
// ===== library types =====

TYPE "ecco"
   STRUCT
      test : Bool;
      "type" : Byte;
      copy : String;
   END_STRUCT;
END_TYPE

FUNCTION_BLOCK "FB-Tipo"   // FB1, LAD
{ S7_Optimized_Access := 'TRUE' }
VERSION : 0.1
BEGIN

REGION Network 1
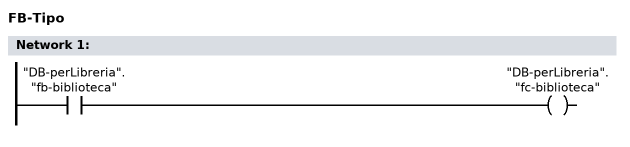
   RUNG wire#powerrail
      Contact( "DB-perLibreria"."fb-biblioteca" )
      Coil( "DB-perLibreria"."fc-biblioteca" )
   END_RUNG
   // the same network as SCL:
   "DB-perLibreria"."fc-biblioteca" := "DB-perLibreria"."fb-biblioteca";
END_REGION
END_FUNCTION_BLOCK

FUNCTION "FC-Tipo" : Void   // FC1, LAD
{ S7_Optimized_Access := 'TRUE' }
VERSION : 0.1
BEGIN

REGION Network 1
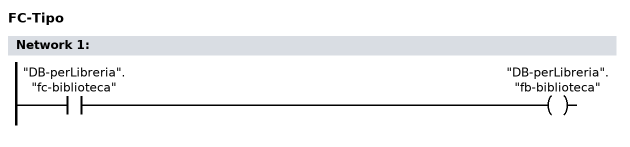
   RUNG wire#powerrail
      Contact( "DB-perLibreria"."fc-biblioteca" )
      Coil( "DB-perLibreria"."fb-biblioteca" )
   END_RUNG
   // the same network as SCL:
   "DB-perLibreria"."fb-biblioteca" := "DB-perLibreria"."fc-biblioteca";
END_REGION
END_FUNCTION

// ===== library: MasterCopy "DB-inLibreria" =====

DATA_BLOCK "DB-perLibreria"   // DB2
{ S7_Optimized_Access := 'TRUE' }
VERSION : 0.1
   VAR
      "fb-biblioteca" : Bool;
      "fc-biblioteca" : Bool;
      prova : "ecco";
   END_VAR
BEGIN
END_DATA_BLOCK

// ===== library: MasterCopy "FB-inLibreria" =====

FUNCTION_BLOCK "FB-inLibreria"   // FB1, LAD
{ S7_Optimized_Access := 'TRUE' }
VERSION : 0.1
BEGIN

REGION Network 1
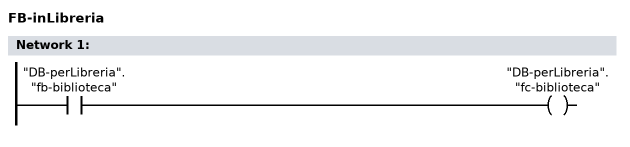
   RUNG wire#powerrail
      Contact( "DB-perLibreria"."fb-biblioteca" )
      Coil( "DB-perLibreria"."fc-biblioteca" )
   END_RUNG
   // the same network as SCL:
   "DB-perLibreria"."fc-biblioteca" := "DB-perLibreria"."fb-biblioteca";
END_REGION
END_FUNCTION_BLOCK

// ===== library: MasterCopy "FC-inLibreria" =====

FUNCTION "FC-inLibreria" : Void   // FC1, LAD
{ S7_Optimized_Access := 'TRUE' }
VERSION : 0.1
BEGIN

REGION Network 1
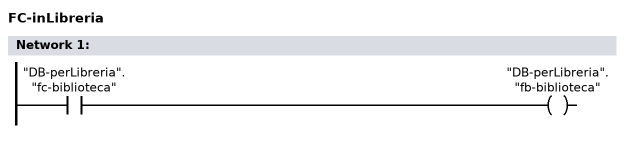
   RUNG wire#powerrail
      Contact( "DB-perLibreria"."fc-biblioteca" )
      Coil( "DB-perLibreria"."fb-biblioteca" )
   END_RUNG
   // the same network as SCL:
   "DB-perLibreria"."fb-biblioteca" := "DB-perLibreria"."fc-biblioteca";
END_REGION
END_FUNCTION

(* ===== HMI "HiddenHmiRTDeviceFaceplateTypes" =====

HMI tags "95890b74-8631-423c-a1c7-cb7e41fdb394"
   "Interface_Tag_1" : bcce95c2-ab17-4d1c-bea8-aafee6094bf9, internal
*)